FUNCTION_BLOCK TimeTicker (* Composite FB wrapping other FBs *)
  (* Standard: 61499-2 *)
  (* Version 1.0, 2026-08-15, franz *)
  PACKAGE adapter::events::TimeOut;
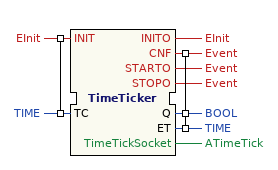
  EVENT_INPUT
    INIT : EInit WITH TC; (* Initialization Request *)
  END_EVENT
  EVENT_OUTPUT
    INITO : EInit; (* Initialization Confirm *)
    CNF WITH Q, ET; (* Reports the current Q/ET on every tick *)
    STARTO;
    STOPO;
  END_EVENT
  VAR_INPUT
    TC : TIME := T#200ms; (* cycleTime *)
  END_VAR
  VAR_OUTPUT
    Q : BOOL; (* Output *)
    ET : TIME; (* Elapsed time *)
  END_VAR
  PLUGS
    TimeTickSocket : adapter::events::TimeOut::ATimeTick;
  END_PLUGS
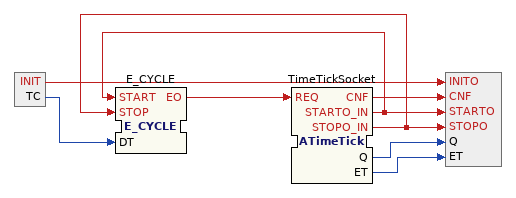
  FBS
    E_CYCLE : iec61499::events::E_CYCLE;
  END_FBS
  EVENT_CONNECTIONS
    E_CYCLE.EO TO TimeTickSocket.REQ;
    INIT TO INITO;
    TimeTickSocket.CNF TO CNF;
    TimeTickSocket.STARTO_IN TO STARTO;
    TimeTickSocket.STOPO_IN TO STOPO;
    TimeTickSocket.STARTO_IN TO E_CYCLE.START;
    TimeTickSocket.STOPO_IN TO E_CYCLE.STOP;
  END_CONNECTIONS
  DATA_CONNECTIONS
    TC TO E_CYCLE.DT;
    TimeTickSocket.Q TO Q;
    TimeTickSocket.ET TO ET;
  END_CONNECTIONS
END_FUNCTION_BLOCK
